FUNCTION_BLOCK FB_PWM
VAR_INPUT
	En: BOOL;
	bEnable: BOOL;                  // Enable PWM alg
	iBlockSampleTimeMicroS: DINT;   // How often this block is called 
	iProcessSampleTimeMicroS: DINT; // Pwm cycle time. iProcessSampleTimeMicroS >> iBlockSampleTimeMicroS to get a good PWM resolution
 	iDecimalPoint: INT;             // At which decimal should teh pwm take place
	fInput: LREAL;                  // Input process value (that will be PWM:ed) 
	// PWM type:
	// Optimized: The low and high values are as ebenly distibuted in time as possible
	// Simple:    Either the low or high values are output first then the other (depending on bPromoteHigh bit)
	ePwmType:E_PWM_TYPE:=E_PWM_TYPE.OPTIMIZED;  
	bPromoteHigh:BOOL:=TRUE; // Only used in simple mode.
END_VAR
VAR_OUTPUT
	EnO: BOOL;
	fOutput: LREAL;
	fOutputError:LREAL:=0;  // Esitmated error of the PWM alg.
END_VAR
VAR
	iNumCycles: DINT;
	iBase: DINT;
	fDecimals: LREAL;
	i: INT;
	iDecimalGain: DINT;
	fOutputHigh: LREAL;
	iHighCycles: DINT;
	iLowCycles: DINT;
	fOutputLow: LREAL;
	iCycleCounter: DINT;
	iLowCounter: INT;
	iHighCounter: INT;
	fActualPWM: LREAL;
	fSetpointPWM: LREAL;
	fInputOld:LREAL:=0;
END_VAR

// Function: PWM block to be used to enhance resolution of signals
//
// Usefull for instance when a ethercat slave communicates with ints and you need 
// higher precision than the int provides. The desired input value are then PWM so that the
// average over processSampleTime is as close as possile to the desired value.
// Block can execute in three different modes:
//   OPTIMIZED: The low and high values are as evently as possible distributed over time
//   SIMPLE:    All high or low values are output first then the other (depending on bPromoteHigh bit)
//   NONE:      Output is same as input (no PWM)
//
// Note: Average resolution will be higher on the cost of sample rate
// Note: Error of PWM alg can be seen in fOutputError
//
// Example: fInput = 23.33333333, iDecimalpoint=3  ==>
//            fOutput will be pulse width modulated with the two discrete values: 23.333 and 23.334
//            in 33% of iProcessSampleTimeMicroS fOutput will be 23.333 and
//            in 67% of iProcessSampleTimeMicroS fOutput will be 23.334
//
// Author: Anders Sandström 2018
//
IF bEnable THEN
  IF(fInput<>fInputOld) THEN // New input value
    iNumCycles:=iProcessSampleTimeMicroS/iBlockSampleTimeMicroS; //71 if 71ms and 1ms
	iDecimalGain:=1;
	FOR i:=1 TO iDecimalPoint DO
      iDecimalGain:=iDecimalGain*10; //10000 if iDecimalpoint is 4
	END_FOR
	iBase:=TRUNC(fInput*iDecimalGain); //=900004 if fOverride=90.00045
    fDecimals:=fInput*iDecimalGain-iBase; //=0.5 if fOverride=90.00045
	iHighCycles:=LREAL_TO_INT(iNumCycles*fDecimals);
    iLowCycles:=iNumCycles-iHighCycles;
    fOutputLow:=DINT_TO_LREAL(iBase)/iDecimalGain; //90.0004
    fOutputHigh:=DINT_TO_LREAL(iBase+1)/iDecimalGain; //90.0005
	iCycleCounter:=0;
	iLowCounter:=0;
	iHighCounter:=0;
	fOutputError:=(fDecimals-DINT_TO_LREAL(iHighCycles)/DINT_TO_LREAL(iNumCycles))/iDecimalGain;
	fSetpointPWM:=DINT_TO_LREAL(iHighCycles)/DINT_TO_LREAL(iLowCycles+iHighCycles);
    END_IF

    IF iCycleCounter > iNumCycles THEN
	  iCycleCounter:=0;
	  iLowCounter:=0;
	  iHighCounter:=0;	
    END_IF
    iCycleCounter:=iCycleCounter+1;
	
  CASE ePwmType OF
	E_PWM_TYPE.OPTIMIZED:  // Distribute low and high evenly in time
       IF iLowCycles > 0 THEN
	     IF iHighCycles > 0 THEN
	       //Both high and low should be output during the period
	       IF iLowCounter = 0 THEN
		     fOutput:=fOutputLow;
		     iLowCounter:=iLowCounter+1;
	       ELSE
	         IF iHighCounter = 0 THEN
		       fOutput:=fOutputHigh;
		       iHighCounter:=iHighCounter+1;
	         ELSE //both counters is atleast 1
		       fActualPWM:= DINT_TO_LREAL(iHighCounter)/DINT_TO_LREAL(iLowCounter+iHighCounter);
		       IF fActualPWM>fSetpointPWM THEN
		         fOutput:=fOutputLow;
		         iLowCounter:=iLowCounter+1;
		       ELSE
                 fOutput:=fOutputHigh;
		         iHighCounter:=iHighCounter+1;
		       END_IF				
	        END_IF				
	      END_IF
        ELSE		
	      fOutput:=fOutputLow;
	      iLowCounter:=iLowCounter+1;
        END_IF
      ELSE
        fOutput:=fOutputHigh;
	    iHighCounter:=iHighCounter+1;
      END_IF
	  
    E_PWM_TYPE.SIMPLE:  // Take all low or high first then the other
	  IF bPromoteHigh THEN  // All high first
        IF iHighCounter < iHighCycles THEN
          iHighCounter:=iHighCounter+1;
		  fOutput:=fOutputHigh;
		ELSE
		  iLowCounter:=iLowCounter+1;
		  fOutput:=fOutputLow;
        END_IF
	  ELSE                  // All low first
        IF iLowCounter < iLowCycles THEN
          iLowCounter:=iLowCounter+1;
		  fOutput:=fOutputLow;
		ELSE
		  iHighCounter:=iHighCounter+1;
		  fOutput:=fOutputHigh;
        END_IF
		  
	  END_IF
	E_PWM_TYPE.NONE:    // Output same as input
	  fOutput:=fInput;
	  iCycleCounter:=0;
	  iLowCounter:=0;
	  iHighCounter:=0;	
	END_CASE
    
ELSE	
	fOutput:=fInput;	
END_IF
fInputOld:=fInput;

END_FUNCTION_BLOCK

(* stored: Version 1.1.0.1, ProductVersion 3.1.4024.0
   POU FB_PWM: Id {329fc295-5889-41aa-b7e1-38a034502569}, SpecialFunc None *)
